(* CODESYS project GlobalVariables.export

Project tree, tasks and I/O mapping:
  GlobalVariables/
    global variables Variables
*)

// GlobalVariables/Variables
{attribute 'qualified_only'}
//{attribute 'conditionalshow'}
//{attribute 'conditionalshow' := 'SomeText'}
//{attribute 'hide'}
VAR_GLOBAL
	g_iDummy : INT; /// This is a dummy global variable
END_VAR
